PROGRAM MAIN
VAR
	(*Design Pattern Blocks *)
	fbPublisher 	: FB_Publisher;
	fbSubscriber 	: ARRAY[1..Param.MaxSubscribers] OF FB_Subscriber;
	
	(* UI Values *)
	AddSub			: ARRAY[1..Param.MaxSubscribers] OF BOOL;
	DeleteSub		: ARRAY[1..Param.MaxSubscribers] OF BOOL;
	i				: INT;
END_VAR

fbPublisher();

FOR i := 1 TO Param.MaxSubscribers DO
	
	IF (AddSub[i]) THEN
		fbPublisher.AddSubscriber(fbSubscriber[i]);
		AddSub[i] := FALSE;
	END_IF

	IF (DeleteSub[i]) THEN
		fbPublisher.RemoveSubscriber(fbSubscriber[i]);
		DeleteSub[i] := FALSE;
	END_IF
	
END_FOR

END_PROGRAM

(* stored: Version 1.1.0.1, ProductVersion 3.1.4022.18
   POU MAIN: Id {7fd8069f-ab2c-4ed6-9213-ca32eb9447ba}, SpecialFunc None *)
